FUNCTION_BLOCK _ArrayDatatype_2D_TestSuite EXTENDS TcUnit.FB_TestSuite
VAR
END_VAR

TestAddress();
TestBaseDatatype();
TestClearReference();
TestClone();
TestTypeNameReturnsExpected();
TestIdentifierReturnsExpected();
TestLength();
TestLowerBoundD1();
TestLowerBoundD2();
TestLowerBoundWithInvalidDimention();
TestMakeReferenceToFollowsReference();
TestMakeReferenceToUpdatesReference();
TestSize();
TestSerializeTypeWith();
TestSerializeWith();
TestTryDeserializeFrom();
TestTryGetElementAsDatatypeWithInvalidDimentionTooBig();
TestTryGetElementAsDatatypeWithInvalidDimentionTooSmall();
TestTryMakeReferenceToFollowsReference();
TestTryMakeReferenceToUpdatesReference();
TestUpperBoundD1();
TestUpperBoundD2();
TestUpperBoundWithInvalidDimention();
TestValueReturnsExpectedAfterChange();

METHOD PUBLIC TestAddress
VAR
    _type : _Array0to1_0to2OfBool;
    notExpected : PVOID := 0;
    actual : PVOID;
END_VAR
TEST('TestAddress');

actual := _type.Address;

AssertFalse(
    Condition := (notExpected = actual),
    Message := 'Type did not return a valid address.'
);

TEST_FINISHED();
END_METHOD

METHOD PUBLIC TestBaseDatatype
VAR
    _type : _Array0to1_0to2OfBool;
    expected : T_MAXSTRING := 'BOOL';
    actual : T_MAXSTRING;
END_VAR
TEST('TestBaseDatatype');

actual := _type.BaseDatatype.TypeName;

AssertEquals_STRING(
    Expected := expected,
    Actual := actual,
    Message := 'Type did not return the correct base type'
);

TEST_FINISHED();
END_METHOD

METHOD PUBLIC TestClearReference
VAR
    _type : _Array0to1_0to2OfBool;
	target : ARRAY [0..1,0..2] OF BOOL;
    expected : ARRAY [0..1,0..2] OF BOOL := [FALSE, FALSE, FALSE, FALSE, FALSE, FALSE];
    actual : ARRAY [0..1,0..2] OF BOOL;
END_VAR
TEST('TestClearReference');

_type.MakeReferenceTo(target);
_type.ClearReference();
target[0,0] := TRUE;

actual := _type.Value;

AssertEquals(
    Expected := expected,
    Actual := actual,
    Message := 'Value incorrectly followed target change'
);

TEST_FINISHED();
END_METHOD

METHOD PUBLIC TestClone
VAR
    _type : _Array0to1_0to2OfBool;
	clone : I_Datatype;
	isValidClone : BOOL;
	compareResult : DINT;
END_VAR
TEST('TestClone');

clone := _type.Clone();

isValidClone := clone <> 0;

IF isValidClone THEN
	compareResult := memcmp(_type.Address, clone.Address, clone.Size);
END_IF

AssertTrue(
	Condition := isValidClone,
	Message := 'Clone did not produce a clone'
);

AssertEquals_DINT(
	Expected := 0,
    Actual := compareResult,
    Message := 'Clone did not return a valid clone.'
);

clone.Dispose();

TEST_FINISHED();
END_METHOD

METHOD PUBLIC TestIdentifierReturnsExpected
VAR
    _type : _Array0to1_0to2OfBool;
    expected : STRING := 'ARRAY [0..1,0..2] OF BOOL';
    actual : STRING;
END_VAR
TEST('TestIdentifierReturnsExpected');

actual := _type.Identifier;

AssertEquals_STRING(
    Expected := expected,
    Actual := actual,
    Message := 'Type did not return correct iec type.'
);

TEST_FINISHED();
END_METHOD

METHOD PUBLIC TestLength
VAR
    _type : _Array0to1_0to2OfBool;
    expected : UDINT := 6;
    actual : UDINT;
END_VAR
TEST('TestLength');

actual := _type.Length;

AssertEquals_UDINT(
    Expected := Expected,
    Actual := actual,
    Message := 'Type did not return the correct array length.'
);

TEST_FINISHED();
END_METHOD

METHOD PUBLIC TestLowerBoundD1
VAR
    _type : _Array0to1_0to2OfBool;
    expected : DINT := 0;
    actual : DINT;
	ok : BOOL;
END_VAR
TEST('TestLowerBoundD1');

ok := _type.TryGetLowerBound(1, actual);

AssertTrue(
    Condition := ok,
    Message := 'Type did not indicate that lower bound was possible to retreive.'
);

AssertEquals_DINT(
    Expected := Expected,
    Actual := actual,
    Message := 'Type did not return the correct array lower bound.'
);

TEST_FINISHED();
END_METHOD

METHOD PUBLIC TestLowerBoundD2
VAR
    _type : _Array0to1_0to2OfBool;
    expected : DINT := 0;
    actual : DINT;
	ok : BOOL;
END_VAR
TEST('TestLowerBoundD2');

ok := _type.TryGetLowerBound(2, actual);

AssertTrue(
    Condition := ok,
    Message := 'Type did not indicate that lower bound was possible to retreive.'
);

AssertEquals_DINT(
    Expected := Expected,
    Actual := actual,
    Message := 'Type did not return the correct array lower bound.'
);

TEST_FINISHED();
END_METHOD

METHOD PUBLIC TestLowerBoundWithInvalidDimention
VAR
    _type : _Array0to1_0to2OfBool;
    actual : DINT;
	result : BOOL;
END_VAR
TEST('TestLowerBoundWithInvalidDimention');

result := _type.TryGetLowerBound(100, actual);

AssertFalse(
    Condition := result,
    Message := 'Type did not indicate that the dimention was invalid'
);

TEST_FINISHED();
END_METHOD

METHOD PUBLIC TestMakeReferenceToFollowsReference
VAR
	_type : _Array0to1_0to2OfBool;
	target : ARRAY [0..1,0..2] OF BOOL;
    expected : ARRAY [0..1,0..2] OF BOOL := [FALSE, TRUE, FALSE, TRUE, FALSE, FALSE];
    actual : ARRAY [0..1,0..2] OF BOOL;
END_VAR
TEST('TestMakeReferenceToFollowsReference');

_type.MakeReferenceTo(target);
target[0,1] := TRUE;
target[1,0] := TRUE;

actual := _type.Value;

AssertEquals(
    Expected := expected,
    Actual := actual,
    Message := 'Value did not follow target change'
);

TEST_FINISHED();
END_METHOD

METHOD PUBLIC TestMakeReferenceToUpdatesReference
VAR
	_type : _Array0to1_0to2OfBool;
	target : ARRAY [0..1,0..2] OF BOOL;
    expected : ARRAY [0..1,0..2] OF BOOL := [FALSE, TRUE, FALSE, TRUE, FALSE, FALSE];
    actual : ARRAY [0..1,0..2] OF BOOL;
END_VAR
TEST('TestMakeReferenceToUpdatesReference');

_type.MakeReferenceTo(target);
_type.Value[0,1] := TRUE;
_type.Value[1,0] := TRUE;

actual := target;

AssertEquals(
    Expected := expected,
    Actual := actual,
    Message := 'Value did not update target'
);

TEST_FINISHED();
END_METHOD

METHOD PUBLIC TestSerializeTypeWith
VAR
    _type : _Array0to1_0to2OfBool;
    serializer : JsonSerializer;
    expected : STRING(1000) := '{"typeName":"ARRAY","identifier":"ARRAY [0..1,0..2] OF BOOL","baseType":{"typeName":"BOOL"}}';
    actual : STRING(1000);
END_VAR
TEST('TestSerializeTypeWith');

serializer.Reset();
_type.SerializeTypeWith(serializer);
serializer.TryGetSerializedData(ADR(actual), SIZEOF(actual));

AssertEquals_STRING(
    Expected := expected,
    Actual := actual,
    Message := 'Serialization of type did not return correct string.'
);

TEST_FINISHED();
END_METHOD

METHOD PUBLIC TestSerializeWith
VAR
    _type : _Array0to1_0to2OfBool;
    serializer : JsonSerializer;
    expected : STRING(500) := '[[false,true,false],[true,false,false]]';
    actual : STRING(500);
END_VAR
TEST('TestSerializeWith');

_type.Value[0,1] := TRUE;
_type.Value[1,0] := TRUE;

serializer.Reset();
_type.SerializeWith(serializer);
serializer.TryGetSerializedData(ADR(actual), SIZEOF(actual));

AssertEquals_STRING(
    Expected := expected,
    Actual := actual,
    Message := 'Serialization of type data did not return correct string.'
);

TEST_FINISHED();
END_METHOD

METHOD PUBLIC TestSize
VAR
    _type : _Array0to1_0to2OfBool;
	example : ARRAY [0..1,0..2] OF BOOL;
    expected : UDINT := SIZEOF(example);
    actual : UDINT;
END_VAR
TEST('TestSize');

actual := _type.Size;

AssertEquals_UDINT(
    Expected := Expected,
    Actual := actual,
    Message := 'Type did not return the correct size.'
);

TEST_FINISHED();
END_METHOD

METHOD PUBLIC TestTryDeserializeFrom
VAR
    deserializer : JsonDeserializer;
    feedback : DeserializerFeedback;
    json : STRING(500) := '[[false,true,false],[true,false,false]]';
    _type : _Array0to1_0to2OfBool;
    expected :  ARRAY [0..1,0..2] OF BOOL := [FALSE, TRUE, FALSE, TRUE, FALSE, FALSE];
    actual : ARRAY [0..1,0..2] OF BOOL;
 END_VAR
TEST('TestTryDeserializeFrom');

deserializer.Reset();
deserializer.TryLoad(json);
_type.TryDeserializeFrom(Deserializer, Feedback);

actual := _type.Value;

AssertEquals(
    Expected := expected,
    Actual := actual,
    Message := 'Type did not deserialize correctly.'
);

TEST_FINISHED();
END_METHOD

METHOD PUBLIC TestTryGetElementAsDatatypeWithInvalidDimentionTooBig
VAR
    _type : _Array0to1_0to2OfBool;
    actual : I_Datatype;
	result : BOOL;
END_VAR
TEST('TestTryGetElementAsDatatypeWithInvalidDimentionTooBig');

result := _type.TryGetElementAsDatatypeByIndex(0,3, actual);

AssertFalse(
    Condition := result,
    Message := 'Type did not indicate that the dimention was invalid'
);

TEST_FINISHED();
END_METHOD

METHOD PUBLIC TestTryGetElementAsDatatypeWithInvalidDimentionTooSmall
VAR
    _type : _Array0to1_0to2OfBool;
    actual : I_Datatype;
	result : BOOL;
END_VAR
TEST('TestTryGetElementAsDatatypeWithInvalidDimentionTooSmall');

result := _type.TryGetElementAsDatatypeByIndex(-1, 0, actual);

AssertFalse(
    Condition := result,
    Message := 'Type did not indicate that the dimention was invalid'
);

TEST_FINISHED();
END_METHOD

METHOD PUBLIC TestTryMakeReferenceToFollowsReference
VAR
    _type : _Array0to1_0to2OfBool;
	target : _Array0to1_0to2OfBool;
    expected : ARRAY [0..1,0..2] OF BOOL := [FALSE, TRUE, FALSE, TRUE, FALSE, FALSE];
    actual :  ARRAY [0..1,0..2] OF BOOL;
END_VAR
TEST('TestTryMakeReferenceToFollowsReference');

_type.TryMakeReferenceTo(target);
target.Value[0,1] := TRUE;
target.Value[1,0] := TRUE;

actual := _type.Value;

AssertEquals(
    Expected := expected,
    Actual := actual,
    Message := 'Value did not follow target change'
);

TEST_FINISHED();
END_METHOD

METHOD PUBLIC TestTryMakeReferenceToUpdatesReference
VAR
    _type : _Array0to1_0to2OfBool;
	target : _Array0to1_0to2OfBool;
    expected : ARRAY [0..1,0..2] OF BOOL := [FALSE, TRUE, FALSE, TRUE, FALSE, FALSE];
    actual : ARRAY [0..1,0..2] OF BOOL;
END_VAR
TEST('TestTryMakeReferenceToUpdatesReference');

_type.TryMakeReferenceTo(target);
_type.Value[0,1] := TRUE;
_type.Value[1,0] := TRUE;

actual := target.Value;

AssertEquals(
    Expected := expected,
    Actual := actual,
    Message := 'Value did not update target'
);

TEST_FINISHED();
END_METHOD

METHOD PUBLIC TestTypeNameReturnsExpected
VAR
    _type : _Array0to1_0to2OfBool;
    expected : STRING := 'ARRAY';
    actual : STRING;
END_VAR
TEST('TestTypeNameReturnsExpected');

actual := _type.TypeName;

AssertEquals_STRING(
    Expected := expected,
    Actual := actual,
    Message := 'Type did not return correct iec type.'
);

TEST_FINISHED();
END_METHOD

METHOD PUBLIC TestUpperBoundD1
VAR
    _type : _Array0to1_0to2OfBool;
    expected : DINT := 1;
    actual : DINT;
	ok : BOOL;
END_VAR
TEST('TestUpperBoundD1');

ok := _type.TryGetUpperBound(1, actual);

AssertTrue(
    Condition := ok,
    Message := 'Type did not indicate that upper bound was possible to retreive.'
);

AssertEquals_DINT(
    Expected := Expected,
    Actual := actual,
    Message := 'Type did not return the correct array upper bound.'
);

TEST_FINISHED();
END_METHOD

METHOD PUBLIC TestUpperBoundD2
VAR
    _type : _Array0to1_0to2OfBool;
    expected : DINT := 2;
    actual : DINT;
	ok : BOOL;
END_VAR
TEST('TestUpperBoundD2');

ok := _type.TryGetUpperBound(2, actual);

AssertTrue(
    Condition := ok,
    Message := 'Type did not indicate that upper bound was possible to retreive.'
);

AssertEquals_DINT(
    Expected := Expected,
    Actual := actual,
    Message := 'Type did not return the correct array upper bound.'
);

TEST_FINISHED();
END_METHOD

METHOD PUBLIC TestUpperBoundWithInvalidDimention
VAR
    _type : _Array0to1_0to2OfBool;
    actual : DINT;
	result : BOOL;
END_VAR
TEST('TestUpperBoundWithInvalidDimention');

result := _type.TryGetUpperBound(3, actual);

AssertFalse(
    Condition := result,
    Message := 'Type did not indicate that the dimention was invalid'
);

TEST_FINISHED();
END_METHOD

METHOD PUBLIC TestValueReturnsExpectedAfterChange
VAR
    _type : _Array0to1_0to2OfBool;
	value : ARRAY [0..1,0..2] OF BOOL := [FALSE, TRUE, FALSE, TRUE, FALSE, FALSE];
    expected : ARRAY [0..1,0..2] OF BOOL := [FALSE, TRUE, FALSE, TRUE, FALSE, FALSE];
    actual : ARRAY [0..1,0..2] OF BOOL;
END_VAR
TEST('TestValueReturnsExpectedAfterChange');

_type.Value := value;
actual := _type.Value;

AssertEquals(
    Expected := expected,
    Actual := actual,
    Message := 'Expected value not returned after change.'
);

TEST_FINISHED();
END_METHOD

END_FUNCTION_BLOCK

(* stored: Version 1.1.0.1, ProductVersion 3.1.4024.13
   POU _ArrayDatatype_2D_TestSuite: Id {bdd79ff7-68ef-0de7-38db-447d6ed888b1}, SpecialFunc None
   Method TestAddress: Id {1a8b8c0f-f062-090b-33e9-12c3b93016b7}
   Method TestBaseDatatype: Id {28f47fee-1f22-09fb-0ba7-46d39c69b92c}
   Method TestClearReference: Id {4e5cecaa-b2e9-0129-0cc6-22ec73e89e9b}
   Method TestClone: Id {2e927e79-33f2-0211-0a06-0cb3f327e3c2}
   Method TestIdentifierReturnsExpected: Id {1f329c78-e168-0891-3bf0-0d2dda97f077}
   Method TestLength: Id {47f5e7f5-4b90-0c4f-056b-c0bc83184a1e}
   Method TestLowerBoundD1: Id {74a4e143-ef99-0266-195a-5584c075df03}
   Method TestLowerBoundD2: Id {acc18410-b446-0068-019f-27cf22c5bc03}
   Method TestLowerBoundWithInvalidDimention: Id {f611c1d0-62a6-033c-36d7-470ba455d7f9}
   Method TestMakeReferenceToFollowsReference: Id {943516c0-8994-0d02-2e10-423cb9b9b07e}
   Method TestMakeReferenceToUpdatesReference: Id {fadf6ca5-f80d-0fab-3f28-27b4efccd7c0}
   Method TestSerializeTypeWith: Id {7afbb386-ef42-0016-05e9-5b51bd66f5ba}
   Method TestSerializeWith: Id {9c990919-1086-0d55-3f6d-81a59b4955f9}
   Method TestSize: Id {a68d28bd-5319-095d-0fab-599550a6f05f}
   Method TestTryDeserializeFrom: Id {a0aee742-808e-0a66-01e0-90ee70c79bdb}
   Method TestTryGetElementAsDatatypeWithInvalidDimentionTooBig: Id {f782908f-5cc9-02f5-3867-60ebdc644a85}
   Method TestTryGetElementAsDatatypeWithInvalidDimentionTooSmall: Id {1cfe82d8-8775-076c-39d5-ddbd76d46271}
   Method TestTryMakeReferenceToFollowsReference: Id {e17ad897-079b-0d9e-2bd1-7bab700b0547}
   Method TestTryMakeReferenceToUpdatesReference: Id {06b4ed6a-dd42-01de-3780-9248a2e81fc6}
   Method TestTypeNameReturnsExpected: Id {8f2ca238-0775-0249-063c-c48ae7896e8c}
   Method TestUpperBoundD1: Id {003b6f21-8c80-0650-0d7b-900110673546}
   Method TestUpperBoundD2: Id {c6205229-9a01-0830-3ed3-6ee746a5b010}
   Method TestUpperBoundWithInvalidDimention: Id {f807d611-59b6-04ee-0623-bf62de68509c}
   Method TestValueReturnsExpectedAfterChange: Id {064fef37-ac3f-0b61-1505-3eab0eae3634} *)
